// TIA Portal V17 export
// export: Created 2023-12-09T21:24:40.0955692Z, ExportSetting WithDefaults, DisplayName Totally Integrated Automation Portal, DisplayVersion V17, DisplayName TIA Portal Openness, DisplayVersion V17, DisplayName TIA Portal Teamcenter Gateway, DisplayVersion V17, DisplayName TIA Portal Version Control Interface, DisplayVersion V17, DisplayName STEP 7 Professional, DisplayVersion V17, DisplayName STEP 7 Safety, DisplayVersion V17, DisplayName WinCC Advanced / Unified PC, DisplayVersion V17
DATA_BLOCK "TSEND_C_DB"   // DB5
// stored: AutoNumber true, InstanceOfName TSEND_C, OfSystemLibElement TSEND_C, OfSystemLibVersion 2.1
"TSEND_C"
   // VAR_INPUT
   //    REQ : Bool;
   //    CONT : Bool;
   //    LEN : UInt;
   // END_VAR
   // VAR_OUTPUT
   //    DONE : Bool;
   //    BUSY : Bool;
   //    ERROR : Bool;
   //    STATUS : Word;
   // END_VAR
   // VAR_IN_OUT
   //    CONNECT : TCON_Param;
   //    DATA : Variant;
   //    COM_RST : Bool;
   // END_VAR
   // VAR
   //    sb_FIRSTSTART : Bool;
   //    sb_REQ : Bool;
   //    sb_STARTFB : Bool;
   //    sb_CON_EST : Bool;
   //    sb_COMRST : Bool;
   //    si_STATE : UInt;
   //    si_JOB : UInt;
   //    sw_ConID : CONN_OUC;
   //    s_TCON { S7_SetPoint := 'True'} : TCON;
   //    s_TDISCON { S7_SetPoint := 'True'} : TDISCON;
   //    s_TSEND { S7_SetPoint := 'True'} : TSEND;
   // END_VAR
BEGIN
END_DATA_BLOCK
